// Mitsubishi GX Works2 project: PLC_V2_5.5   PLC: FX3G

// global labels: Global1
VAR_GLOBAL
  D_1101 AT D1101 : REAL;
  D_1103 AT D1103 : REAL;
  D_1105 AT D1105 : REAL;
  D_1107 AT D1107 : REAL;
  D_1109 AT D1109 : REAL;
END_VAR
VAR_GLOBAL CONSTANT
  E_0 : REAL;
  E_5 : REAL := 5.0;
  E_6 : REAL := 6.0;
  E_10 : REAL := 10.0;
  RaspberryReg : REAL := 280.0;
  LemonReg : REAL := 455.0;
  StabReg : REAL := 105.0;
  BearsReg : REAL := 28.0;
  RaspberryTreat : REAL := 385.0;
  LemonTreat : REAL := 665.0;
  StabTreat : REAL := 210.0;
  BearsTreat : REAL := 70.0;
END_VAR
VAR_GLOBAL
  D_8280 AT D8280 : INT;
  M_0 AT M0 : BOOL;
  M_2 AT M2 : BOOL;
  M_3 AT M3 : BOOL;
  M_100 AT M100 : BOOL;
  M_101 AT M101 : BOOL;
  M_102 AT M102 : BOOL;
  M_200 AT M200 : BOOL;
  M_201 AT M201 : BOOL;
  M_202 AT M202 : BOOL;
  M_203 AT M203 : BOOL;
  M_220 AT M220 : BOOL;
  M_221 AT M221 : BOOL;
  M_222 AT M222 : BOOL;
  M_223 AT M223 : BOOL;
  M_210 AT M210 : BOOL;
  M_211 AT M211 : BOOL;
  M_300 AT M300 : BOOL;
  M_301 AT M301 : BOOL;
  M_400 AT M400 : BOOL;
  M_401 AT M401 : BOOL;
  K_800 : REAL;
  M_302 AT M302 : BOOL;
  M_500 AT M500 : BOOL;
  M_501 AT M501 : BOOL;
  M_502 AT M502 : BOOL;
  M_510 AT M510 : BOOL;
END_VAR
VAR_GLOBAL CONSTANT
  E_1 : REAL := 1.0;
END_VAR
VAR_GLOBAL
  D_1119 AT D1119 : REAL;
  M_60 AT M60 : BOOL;
  M_520 : BOOL;
  M_521 : BOOL;
  M_103 AT M103 : BOOL;
  M_104 AT M104 : BOOL;
  M_105 AT M105 : BOOL;
  M_106 AT M106 : BOOL;
  M_212 AT M212 : BOOL;
  M_213 AT M213 : BOOL;
END_VAR
VAR_GLOBAL CONSTANT
  E_400 : REAL := 400.0;
END_VAR
VAR_GLOBAL
  D_1121 AT D1121 : REAL;
END_VAR

// task Task_01 (event TRUE, interval 0, priority 31): POU_01

PROGRAM POU_01
(* structured ladder/FBD written out as ST: instructions are called as NAME(EN, inputs, outputs); _pN, _eN, _tN stand for wires *)
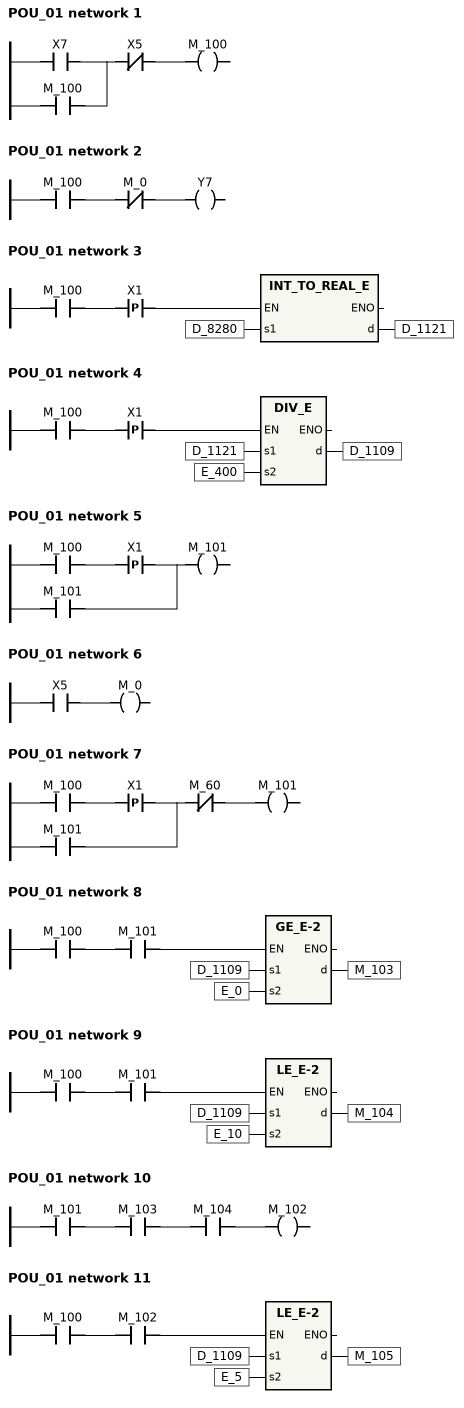
(* network 1 *)
M_100 := (X7 OR M_100) AND NOT X5;
(* network 2 *)
Y7 := M_100 AND NOT M_0;
(* network 3 *)
INT_TO_REAL_E(M_100 AND LDP(TRUE, X1), D_8280, D_1121);
(* network 4 *)
DIV_E(M_100 AND LDP(TRUE, X1), D_1121, E_400, D_1109);
(* network 5 *)
M_101 := (M_100 AND LDP(TRUE, X1)) OR M_101;
(* network 6 *)
M_0 := X5;
(* network 7 *)
M_101 := ((M_100 AND LDP(TRUE, X1)) OR M_101) AND NOT M_60;
(* network 8 *)
GE_E(M_100 AND M_101, D_1109, E_0, M_103);
(* network 9 *)
LE_E(M_100 AND M_101, D_1109, E_10, M_104);
(* network 10 *)
M_102 := M_101 AND M_103 AND M_104;
(* network 11 *)
LE_E(M_100 AND M_102, D_1109, E_5, M_105);
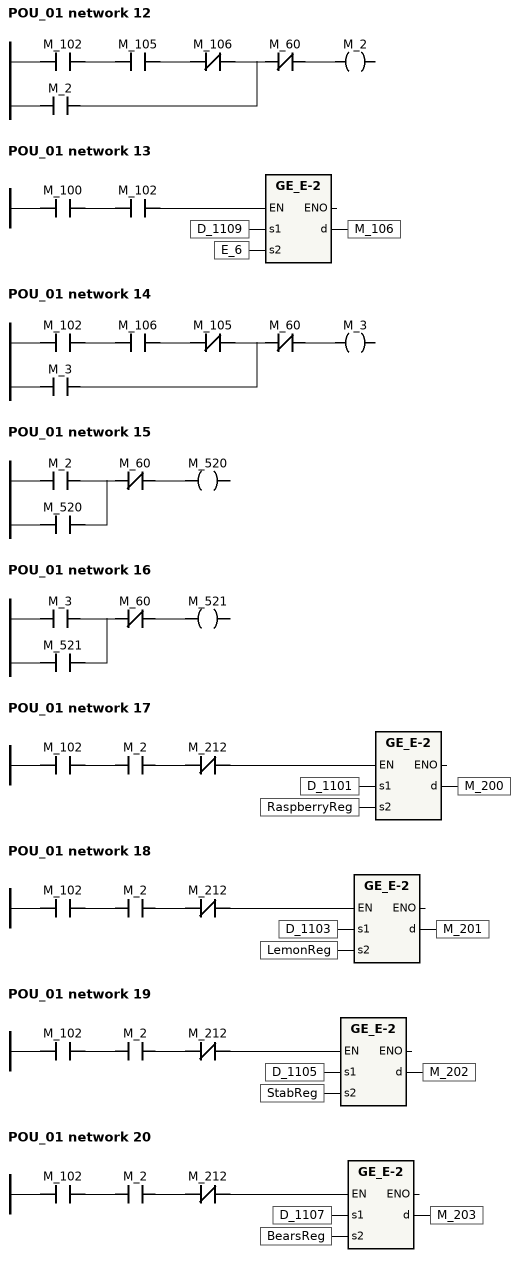
(* network 12 *)
M_2 := ((M_102 AND M_105 AND NOT M_106) OR M_2) AND NOT M_60;
(* network 13 *)
GE_E(M_100 AND M_102, D_1109, E_6, M_106);
(* network 14 *)
M_3 := ((M_102 AND M_106 AND NOT M_105) OR M_3) AND NOT M_60;
(* network 15 *)
M_520 := (M_2 OR M_520) AND NOT M_60;
(* network 16 *)
M_521 := (M_3 OR M_521) AND NOT M_60;
(* network 17 *)
GE_E(M_102 AND M_2 AND NOT M_212, D_1101, RaspberryReg, M_200);
(* network 18 *)
GE_E(M_102 AND M_2 AND NOT M_212, D_1103, LemonReg, M_201);
(* network 19 *)
GE_E(M_102 AND M_2 AND NOT M_212, D_1105, StabReg, M_202);
(* network 20 *)
GE_E(M_102 AND M_2 AND NOT M_212, D_1107, BearsReg, M_203);
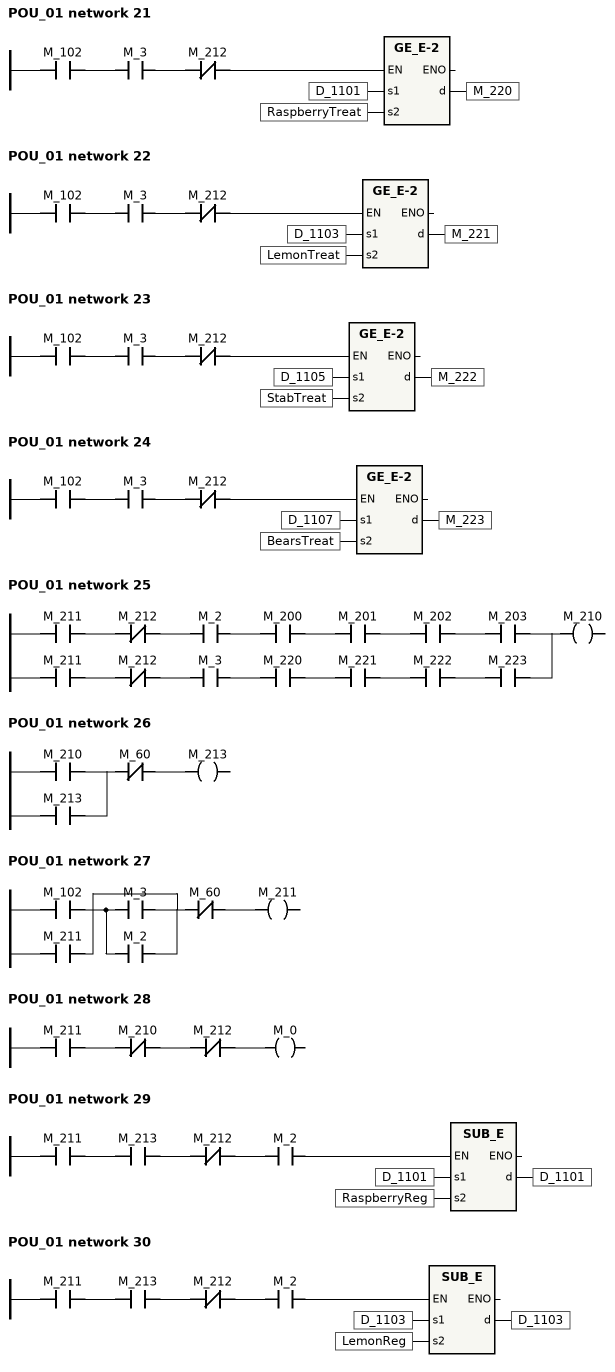
(* network 21 *)
GE_E(M_102 AND M_3 AND NOT M_212, D_1101, RaspberryTreat, M_220);
(* network 22 *)
GE_E(M_102 AND M_3 AND NOT M_212, D_1103, LemonTreat, M_221);
(* network 23 *)
GE_E(M_102 AND M_3 AND NOT M_212, D_1105, StabTreat, M_222);
(* network 24 *)
GE_E(M_102 AND M_3 AND NOT M_212, D_1107, BearsTreat, M_223);
(* network 25 *)
M_210 := (M_211 AND NOT M_212 AND M_2 AND M_200 AND M_201 AND M_202 AND M_203) OR (M_211 AND NOT M_212 AND M_3 AND M_220 AND M_221 AND M_222 AND M_223);
(* network 26 *)
M_213 := (M_210 OR M_213) AND NOT M_60;
(* network 27 *)
M_211 := ((M_102 AND M_3) OR (M_102 AND M_2) OR M_211) AND NOT M_60;
(* network 28 *)
M_0 := M_211 AND NOT M_210 AND NOT M_212;
(* network 29 *)
SUB_E(M_211 AND M_213 AND NOT M_212 AND M_2, D_1101, RaspberryReg, D_1101);
(* network 30 *)
SUB_E(M_211 AND M_213 AND NOT M_212 AND M_2, D_1103, LemonReg, D_1103);
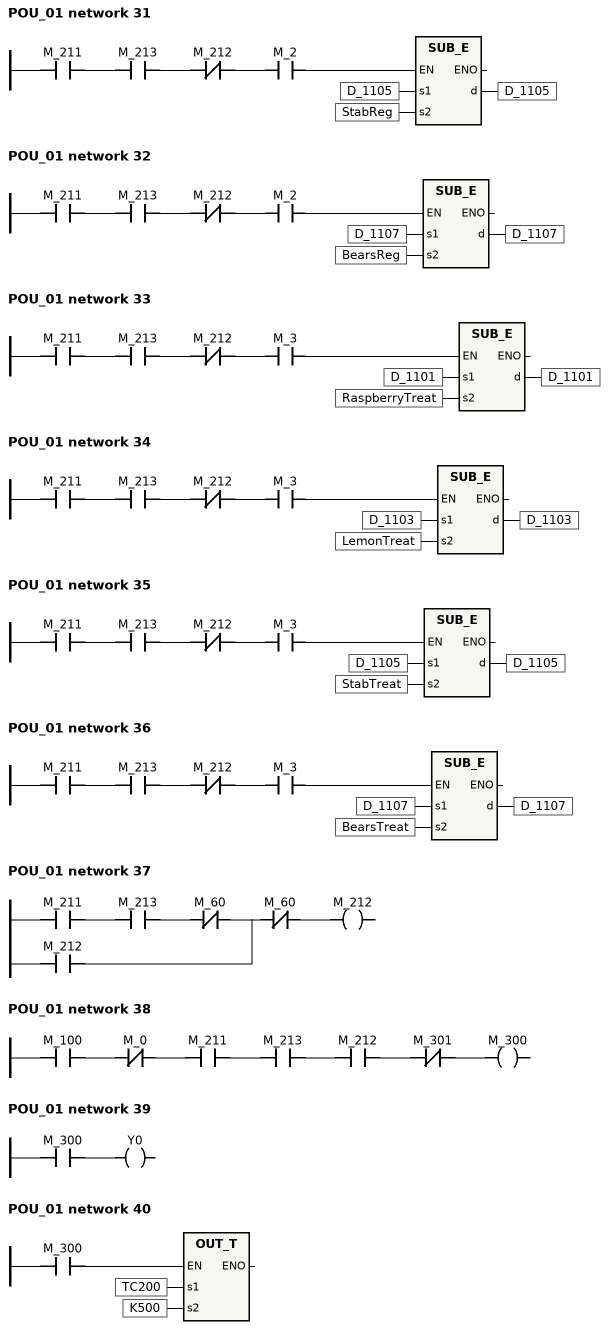
(* network 31 *)
SUB_E(M_211 AND M_213 AND NOT M_212 AND M_2, D_1105, StabReg, D_1105);
(* network 32 *)
SUB_E(M_211 AND M_213 AND NOT M_212 AND M_2, D_1107, BearsReg, D_1107);
(* network 33 *)
SUB_E(M_211 AND M_213 AND NOT M_212 AND M_3, D_1101, RaspberryTreat, D_1101);
(* network 34 *)
SUB_E(M_211 AND M_213 AND NOT M_212 AND M_3, D_1103, LemonTreat, D_1103);
(* network 35 *)
SUB_E(M_211 AND M_213 AND NOT M_212 AND M_3, D_1105, StabTreat, D_1105);
(* network 36 *)
SUB_E(M_211 AND M_213 AND NOT M_212 AND M_3, D_1107, BearsTreat, D_1107);
(* network 37 *)
M_212 := ((M_211 AND M_213 AND NOT M_60) OR M_212) AND NOT M_60;
(* network 38 *)
M_300 := M_100 AND NOT M_0 AND M_211 AND M_213 AND M_212 AND NOT M_301;
(* network 39 *)
Y0 := M_300;
(* network 40 *)
OUT_T(M_300, TC200, K500);
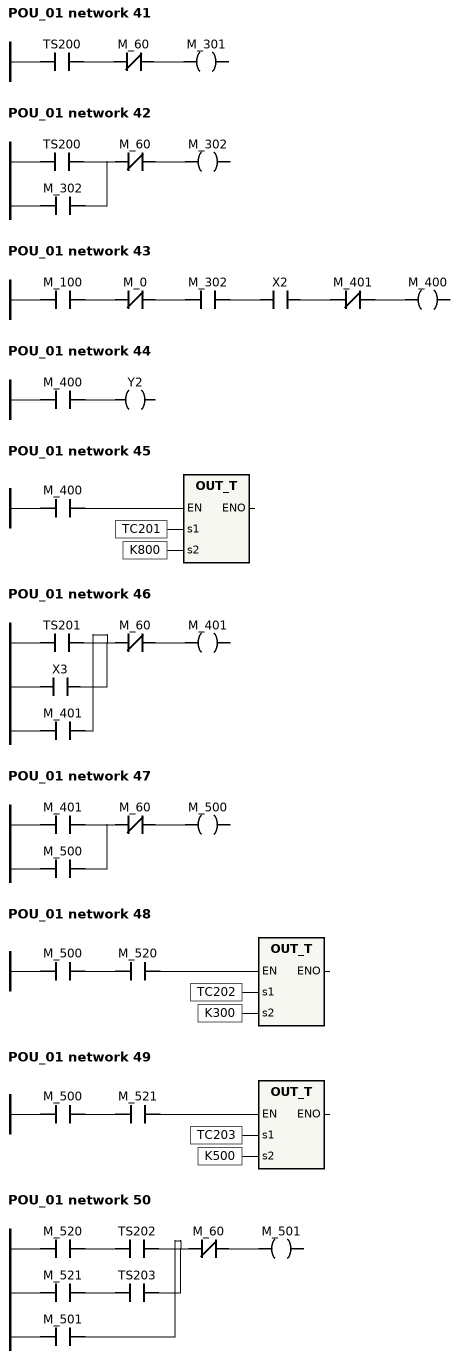
(* network 41 *)
M_301 := TS200 AND NOT M_60;
(* network 42 *)
M_302 := (TS200 OR M_302) AND NOT M_60;
(* network 43 *)
M_400 := M_100 AND NOT M_0 AND M_302 AND X2 AND NOT M_401;
(* network 44 *)
Y2 := M_400;
(* network 45 *)
OUT_T(M_400, TC201, K800);
(* network 46 *)
M_401 := (TS201 OR X3 OR M_401) AND NOT M_60;
(* network 47 *)
M_500 := (M_401 OR M_500) AND NOT M_60;
(* network 48 *)
OUT_T(M_500 AND M_520, TC202, K300);
(* network 49 *)
OUT_T(M_500 AND M_521, TC203, K500);
(* network 50 *)
M_501 := ((M_520 AND TS202) OR (M_521 AND TS203) OR M_501) AND NOT M_60;
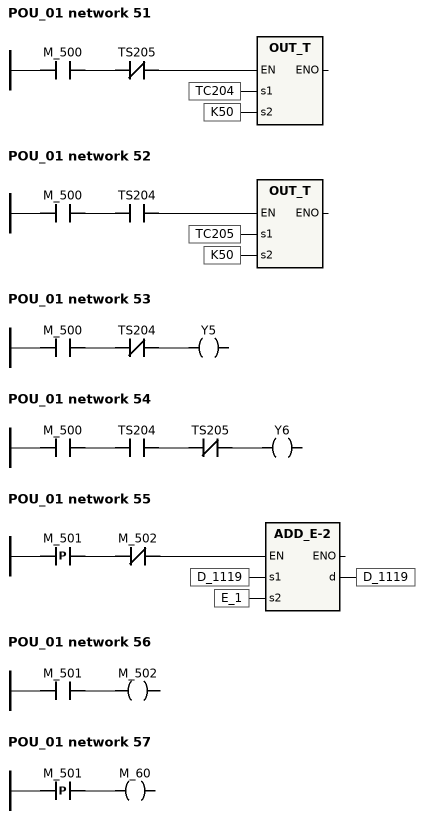
(* network 51 *)
OUT_T(M_500 AND NOT TS205, TC204, K50);
(* network 52 *)
OUT_T(M_500 AND TS204, TC205, K50);
(* network 53 *)
Y5 := M_500 AND NOT TS204;
(* network 54 *)
Y6 := M_500 AND TS204 AND NOT TS205;
(* network 55 *)
ADD_E(LDP(TRUE, M_501) AND NOT M_502, D_1119, E_1, D_1119);
(* network 56 *)
M_502 := M_501;
(* network 57 *)
M_60 := LDP(TRUE, M_501);
END_PROGRAM
